PROGRAM prStation6
VAR
    SolFix : fbSingleSolRy;
    SolUpDown : fbSingleSolRy;
    SolClamp : fbSingleSolRy;
    ErrorState : BOOL;
    Autoflow : INT;
    torqueArrived1 : BOOL;
    torqueArrived2 : BOOL;
    screwL : UINT;
    oldTorqueR : LREAL;
    oldTorqueL : LREAL;
    screwR : UINT;
    TON1 : TON;
    TON2 : TON;
    ScrewLeft : fbScrewFlow;
    ScrewRight : fbScrewFlow;
    TON3 : TON;
END_VAR
VAR_EXTERNAL
    HMIPB_SOL_S5_Fix : BOOL;
    AutoStatus : bool;
    SNR_Index : BOOL;
    RY_Index : BOOL;
    SOL_S5_Fix : BOOL;
    HMIPB_SOL_S5_UpDown : BOOL;
    SOL_S5_UpDown : BOOL;
    HMIPB_SOL_S5_Clamp : BOOL;
    SOL_S5_Clamp : BOOL;
    HMIPB_SOL_S6_Fix : BOOL;
    SOL_S6_Feed : BOOL;
    SOL_S6_Fix : BOOL;
    HMIPB_SOL_S6_UpDown : BOOL;
    SOL_S6_UpDown : BOOL;
    HMIPB_SOL_S6_Clamp : BOOL;
    SOL_S6_Clamp : BOOL;
    Error_PB_Estop1 : BOOL;
    Error_PB_Estop2 : BOOL;
    Error_LS_S6_FixBack : BOOL;
    Error_LS_S6_FixOut : BOOL;
    Error_LS_S6_UpDownBack : BOOL;
    Error_LS_S6_UpDownOut : BOOL;
    IndexData6 : StationRecord;
    SystemReadyStatus : bool;
    MachineRunStatus : bool;
    HMI_ScrewTorque_St5_L : LREAL;
    HMI_ScrewSpeed_St5_L : LREAL;
    HMI_ScrewTorque_St5_R : LREAL;
    HMI_ScrewSpeed_St5_R : LREAL;
    HMIShow_CurrentTorque : ARRAY[0..3] OF LREAL;
    HMIPB_ServoStopAxisLSt5 : BOOL;
    HMIPB_ServoStopAxisRSt5 : BOOL;
    HMIPB_FW_AxisLSt5 : BOOL;
    HMIPB_FW_AxisRSt5 : BOOL;
    ScrewStartFlag : ARRAY[0..3] OF bool;
    HMI_ScrewTorque_St6_R : LREAL;
    HMI_ScrewTorque_St6_L : LREAL;
    HMI_ScrewSpeed_St6_R : LREAL;
    HMI_ScrewSpeed_St6_L : LREAL;
    HMIPB_FW_AxisLSt6 : BOOL;
    HMIPB_FW_AxisRSt6 : BOOL;
    LS_S6_UpDownOut : BOOL;
    LS_S6_UpDownBack : BOOL;
    SNR_S6_R_Check : BOOL;
    HMIPB_RW_AxisRSt6 : BOOL;
    HMIShow_CurrentSpeed : ARRAY[0..3] OF LREAL;
    LS_S6_FixBack : BOOL;
    SNR_S6_L_Check : BOOL;
    HMIPB_RW_AxisLSt6 : BOOL;
    LS_S2_MoveBack : BOOL;
    FeedStartFlag : ARRAY[0..1] OF bool;
    OBJScrewInClip : ARRAY[0..3] OF INT;
END_VAR
VAR_EXTERNAL CONSTANT
    MC_AxisLSt5 : _sAXIS_REF;
    MC_AxisLSt6 : _sAXIS_REF;
    MC_AxisRSt6 : _sAXIS_REF;
END_VAR
VAR_EXTERNAL
    ScrewStartS6LFW : BOOL;
    ScrewStartS6LRW : BOOL;
    ScrewStartS6RFW : BOOL;
    ScrewStartS6RRW : BOOL;
    HMI_BackOutTorque_St6_L : LREAL;
    HMI_BackOutTorque_St6_R : LREAL;
    Error_SNR_S6_L_Feed : BOOL;
    Error_SNR_S6_R_Feed : BOOL;
    HMI_LimitAngle_St6_L : LREAL;
    HMIShow_CurrentPosition : ARRAY[0..3] OF LREAL;
    HMI_LimitAngle_St6_R : LREAL;
    ResetAddress : ARRAY[0..3] OF bool;
    HMI_BackOutAngle_St6_L : LREAL;
    HMI_BackOutAngle_St6_R : LREAL;
    BackoutBusy : ARRAY[0..3] OF BOOL;
    BackoutStart : ARRAY[0..3] OF BOOL;
    HMI_NoScrewAngle_St6_L : LREAL;
    HMI_NoScrewAngle_St6_R : LREAL;
    HMI_Find_St6_L : LINT;
    HMI_Find_St6_R : LINT;
END_VAR
SolFix(
	inPushButton:=HMIPB_SOL_S6_Fix,
	inAutoStatus:=AutoStatus,
	inAutoFlowSet:=Autoflow=2,
	inAutoFlowReset:=Autoflow=4 OR ErrorState,
	inInterLockBack:=TRUE,
	inInterLockOut:=SNR_Index AND NOT(RY_Index),
	outSol=>SOL_S6_Fix);
SolUpDown(
	inPushButton:=HMIPB_SOL_S6_UpDown,
	inAutoStatus:=AutoStatus,
	inAutoFlowSet:=Autoflow=2,
	inAutoFlowReset:=Autoflow=4 OR ErrorState,
	inInterLockBack:=TRUE,
	inInterLockOut:=SNR_Index AND NOT(RY_Index),
	outSol=>SOL_S6_UpDown);
SolClamp(
	inPushButton:=HMIPB_SOL_S6_Clamp,
	inAutoStatus:=AutoStatus,
	inAutoFlowSet:=SOL_S6_UpDown AND LS_S6_UpDownOut AND AutoStatus AND (screwR>=2 AND screwR<20 AND screwL>=2 AND screwL<20),
	inAutoFlowReset:=(LS_S6_UpDownBack AND NOT(SOL_S6_UpDown) AND AutoStatus) OR ErrorState,
	inInterLockBack:=TRUE,
	inInterLockOut:=TRUE,
	outSol=>SOL_S6_Clamp);
TON3(In:=SOL_S6_UpDown AND LS_S6_UpDownOut AND AutoStatus,PT:=t#500ms);
(*************************************************************************************************************)
(*EStOP and Error*)
IF (Error_PB_Estop1 OR Error_PB_Estop2) AND NOT(IndexData6.OKFlag_3[6]) THEN
	IndexData6.NGFlag_3[6]:=TRUE;
	IndexData6.ErrorRecordData[6]:=1;
END_IF;
IF (Error_PB_Estop1 OR Error_PB_Estop2) AND NOT(IndexData6.OKFlag_1[6]) THEN
	IndexData6.NGFlag_1[6]:=TRUE;
	IndexData6.ErrorRecordData[6]:=1;
END_IF;
IF ErrorState AND NOT(IndexData6.OKFlag_3[6]) THEN
	IndexData6.NGFlag_3[6]:=TRUE;
	IndexData6.ErrorRecordData[6]:=2;
END_IF;
IF ErrorState AND NOT(IndexData6.OKFlag_1[6]) THEN
	IndexData6.NGFlag_1[6]:=TRUE;
	IndexData6.ErrorRecordData[6]:=2;
END_IF;
(*本站狀態判斷*)
IF (IndexData6.OKFlag_3[6] OR IndexData6.NGFlag_3[6]) AND
	(IndexData6.OKFlag_1[6] OR IndexData6.NGFlag_1[6])
	THEN
	IndexData6.FinishFlag[6]:=TRUE;
END_IF;
(*前站判斷*)
IF IndexData6.NGFlag_3[3] OR NOT(IndexData6.OKFlag_3[3]) THEN
	IndexData6.NGFlag_3[6]:=TRUE;
END_IF;
IF IndexData6.NGFlag_1[3] OR NOT(IndexData6.OKFlag_1[3]) THEN
	IndexData6.NGFlag_1[6]:=TRUE;
END_IF;
(*異常*)
ErrorState:=
Error_LS_S6_FixBack OR
Error_LS_S6_FixOut OR
Error_LS_S6_UpDownBack OR
Error_LS_S6_UpDownOut;
//*********************************自動********************************************
//****************************power on=0
IF NOT(SystemReadyStatus) OR ErrorState OR Error_PB_Estop1 OR Error_PB_Estop2 OR NOT(AutoStatus) THEN
	Autoflow:=0;
END_IF;
//****************************idle=1
IF AutoFlow=0 AND NOT(NOT(SystemReadyStatus) OR ErrorState OR Error_PB_Estop1 OR Error_PB_Estop2 OR NOT(AutoStatus)) THEN
	AutoFlow:=1;
END_IF;
IF Autoflow=4 AND screwL=1 AND screwR=1 AND LS_S6_FixBack AND LS_S6_UpDownBack THEN
	SOL_S6_Clamp:=FALSE;
	Autoflow:=1;
END_IF;
//****************************定位出,向下,鎖付開始=2
IF AutoFlow=1 AND
	NOT(FeedStartFlag[1]) AND
	NOT(Error_SNR_S6_L_Feed) AND
	NOT(Error_SNR_S6_R_Feed) AND
	NOT(SOL_S6_Feed) AND
	SNR_Index AND
	NOT(RY_Index) AND
	MachineRunStatus AND
	NOT(IndexData6.FinishFlag[6]) THEN
	ScrewStartFlag[2]:=TRUE;
	ScrewStartFlag[3]:=TRUE;
	Autoflow:=2;
END_IF;
//****************************鎖付OK=3
IF Autoflow=2 AND screwL=8 THEN//鎖付OK
	ScrewStartFlag[2]:=FALSE;
	IndexData6.OKFlag_3[6]:=TRUE;
END_IF;
IF Autoflow=2 AND screwL=9999 THEN//鎖付NG
	ScrewStartFlag[2]:=FALSE;
	IndexData6.NGFlag_3[6]:=TRUE;
END_IF;
IF Autoflow=2 AND screwR=8 THEN//鎖付OK
	ScrewStartFlag[3]:=FALSE;
	IndexData6.OKFlag_1[6]:=TRUE;
END_IF;
IF Autoflow=2 AND screwR=9999 THEN//鎖付NG
	ScrewStartFlag[3]:=FALSE;
	IndexData6.NGFlag_1[6]:=TRUE;
END_IF;
IF Autoflow=2 AND IndexData6.FinishFlag[6] THEN
	Autoflow:=3;
END_IF;
//****************************向上,定位回=4
IF Autoflow=3 AND LS_S6_UpDownOut AND NOT(ScrewStartFlag[2]) AND NOT(ScrewStartFlag[3]) THEN
	Autoflow:=4;
END_IF;
IF LS_S6_UpDownOut AND SOL_S6_UpDown AND AutoStatus THEN
	FeedStartFlag[1]:=TRUE;
END_IF;
ScrewLeft(
	inStartFlag:=ScrewStartFlag[2],
	inCheckSensor:=SNR_S6_L_Check,
	inStopFlag:= MC_AxisLSt6.Status.Standstill,
	inBackoutBusy:=BackoutBusy[2],
	inCMDTorque:=HMI_BackOutTorque_St6_L,
	inCMDAddress:=HMI_LimitAngle_St6_L,
	inNoScrewSetAngle:=HMI_NoScrewAngle_St6_L,
	inFindTime:=HMI_Find_St6_L,
	inTorqueValue:=HMIShow_CurrentTorque[2],
	inAddressValue:=HMIShow_CurrentPosition[2],
	outFW=>ScrewStartS6LFW,
	outRW=>ScrewStartS6LRW,
	outBackout=>BackoutStart[2],
	outFlowNo=> screwL,
	outResetAddress=>ResetAddress[2],
	inoutTorque:= HMI_ScrewTorque_St6_L);
ScrewRight(
	inStartFlag:=ScrewStartFlag[3],
	inCheckSensor:=SNR_S6_R_Check,
	inStopFlag:= MC_AxisRSt6.Status.Standstill,
	inBackoutBusy:=BackoutBusy[3],
	inCMDTorque:=HMI_BackOutTorque_St6_R,
	inCMDAddress:=HMI_LimitAngle_St6_R,
	inNoScrewSetAngle:=HMI_NoScrewAngle_St6_R,
	inFindTime:=HMI_Find_St6_R,
	inTorqueValue:=HMIShow_CurrentTorque[3],
	inAddressValue:=HMIShow_CurrentPosition[3],
	outFW=>ScrewStartS6RFW,
	outRW=>ScrewStartS6RRW,
	outBackout=>BackoutStart[3],
	outFlowNo=> screwR,
	outResetAddress=>ResetAddress[3],
	inoutTorque:= HMI_ScrewTorque_St6_R);
END_PROGRAM

FUNCTION fIndexDataChange : BOOL
VAR_EXTERNAL
    IndexData8 : StationRecord;
    IndexData7 : StationRecord;
    IndexData6 : StationRecord;
    IndexData5 : StationRecord;
    IndexData4 : StationRecord;
    IndexData3 : StationRecord;
    IndexData2 : StationRecord;
    IndexData1 : StationRecord;
    IndexData0 : StationRecord;
END_VAR
IndexData8:=IndexData7;
IndexData7:=IndexData6;
IndexData6:=IndexData5;
IndexData5:=IndexData4;
IndexData4:=IndexData3;
IndexData3:=IndexData2;
IndexData2:=IndexData1;
IndexData1:=IndexData0;
END_FUNCTION

FUNCTION_BLOCK fbBowlFeeder
VAR
    AutoFlow : INT;
    TON_Auto1 : TON;
    TON_Auto2 : TON;
    TON_Auto3 : TON;
    tItemNotExistDelayTime : TIME;
    tItemExistTime : TIME;
    tItemNotExistErrorTime : TIME;
END_VAR
VAR_INPUT
    bFullSNR : BOOL;
    iItemNotExistDelayTime : LINT;
    iItemExistTime : LINT;
    iItemNotExistErrorTime : LINT;
END_VAR
VAR_OUTPUT
    bFullRY : BOOL;
    bFullSNRError : BOOL;
END_VAR
VAR_EXTERNAL
    SystemReadyStatus : BOOL;
END_VAR
(******************************************************************
程式:振動筒程序
作者:蔡相偉
版本資訊:v1.0		2016/4/16
******************************************************************)
//時間轉換
tItemNotExistDelayTime:=NanoSecToTime(In:=iItemNotExistDelayTime*100000000);
tItemExistTime:=NanoSecToTime(In:=iItemExistTime*100000000);
tItemNotExistErrorTime:=NanoSecToTime(In:=iItemNotExistErrorTime*100000000);
(*流程*)
(*PowerOn=0*)
IF NOT(SystemReadyStatus) THEN
	AutoFlow:=0;
END_IF;

(*Idle=1*)
IF AutoFlow=0 AND SystemReadyStatus THEN
	AutoFlow:=1;
END_IF;

IF AutoFlow=3 THEN
	AutoFlow:=1;
END_IF;

(*振動筒起振=2*)
TON_Auto1(IN:=AutoFlow=1 AND NOT(bFullSNR) , PT:=tItemNotExistDelayTime);
IF AutoFlow=1 AND TON_Auto1.Q THEN
	AutoFlow:=2;
END_IF;

(*振動筒停振=3*)
TON_Auto2(IN:=AutoFlow=2 AND bFullSNR , PT:=tItemExistTime);
TON_Auto3(IN:=NOT(bFullSNR) AND bFullRY, PT:=tItemNotExistErrorTime);
IF AutoFlow=2 AND TON_Auto2.Q THEN
	AutoFlow:=3;
END_IF;
(******************************************************************)
(*輸出*)
(*振動筒繼電器*)
IF AutoFlow=2 THEN
	bFullRY:=TRUE;
	ELSE
	bFullRY:=FALSE;
END_IF;
(*振動筒滿料異常*)
IF AutoFlow=2 AND (TON_Auto3.Q) THEN
	bFullSNRError:=TRUE;
	ELSE
	bFullSNRError:=FALSE;
END_IF;
END_FUNCTION_BLOCK

FUNCTION_BLOCK fbSingleSolRy
VAR
    solStatus : BOOL;
    R_TRIG1 : R_TRIG;
END_VAR
VAR_INPUT
    inPushButton : BOOL;
    inAutoStatus : BOOL;
    inAutoFlowSet : BOOL;
    inAutoFlowReset : BOOL;
    inInterLockBack : BOOL;
    inInterLockOut : BOOL;
END_VAR
VAR_OUTPUT
    outSol : BOOL;
END_VAR
(*電磁閥*)
R_TRIG1(Clk:=inPushButton AND NOT(inAutoStatus));
(*SET*)
IF ((R_TRIG1.Q AND NOT(solStatus)) OR inAutoFlowSet) AND inInterLockOut THEN
	outSol:=TRUE;
END_IF;
(*RESET*)
IF ((R_TRIG1.Q AND (solStatus)) OR inAutoFlowReset) AND inInterLockBack THEN
	outSol:=FALSE;
END_IF;
(*STATUS*)
solStatus:=outSol;
END_FUNCTION_BLOCK

FUNCTION_BLOCK fbErrorSOL_S
VAR
    TON_1 : TON;
    TON_2 : TON;
END_VAR
VAR_INPUT
    bAutoStatus : BOOL;
    bResetPB : BOOL;
    bSOL : BOOL;
    bBackLS : BOOL;
    bOutLS : BOOL;
END_VAR
VAR_OUTPUT
    bErrorStatus_Back : BOOL;
    bErrorStatus_Out : BOOL;
END_VAR
IF bAutoStatus AND NOT(bResetPB) THEN
	(*歸磁簧開關*)
	TON_1(IN:=(NOT(bSOL) AND NOT(bBackLS)) OR ((bSOL) AND bBackLS), PT:=t#2s);
	IF TON_1.Q THEN
		bErrorStatus_Back:=TRUE;
	END_IF;
	(*出磁簧開關*)
	TON_2(IN:=(NOT(bSOL) AND (bOutLS)) OR ((bSOL) AND NOT(bOutLS)), PT:=t#2s);
	IF TON_2.Q THEN
		bErrorStatus_Out:=TRUE;
	END_IF;
END_IF;
IF bResetPB THEN
	bErrorStatus_Back:=FALSE;
	bErrorStatus_Out:=FALSE;
END_IF;
END_FUNCTION_BLOCK

FUNCTION_BLOCK fbErrorSOL_D
VAR
    TON_1 : TON;
    TON_2 : TON;
END_VAR
VAR_INPUT
    bAutoStatus : BOOL;
    bResetPB : BOOL;
    bBackSOL : BOOL;
    bOutSOL : BOOL;
    bBackLS : BOOL;
    bOutLS : BOOL;
END_VAR
VAR_OUTPUT
    bErrorStatus_Back : BOOL;
    bErrorStatus_Out : BOOL;
END_VAR
IF bAutoStatus AND NOT(bResetPB) THEN
	(*歸磁簧開關*)
	TON_1(IN:=bBackSOL AND NOT(bBackLS), PT:=t#4s);
	IF TON_1.Q THEN
		bErrorStatus_Back:=TRUE;
	END_IF;
	(*出磁簧開關*)
	TON_2(IN:=bOutSOL AND NOT(bOutLS), PT:=t#4s);
	IF TON_2.Q THEN
		bErrorStatus_Out:=TRUE;
	END_IF;
END_IF;
IF bResetPB THEN
	bErrorStatus_Back:=FALSE;
	bErrorStatus_Out:=FALSE;
END_IF;
END_FUNCTION_BLOCK

FUNCTION_BLOCK fbCheckScrew_Clamp
VAR
    R_TRIG1 : R_TRIG;
    R_TRIG2 : R_TRIG;
    F_TRIG1 : F_TRIG;
END_VAR
VAR_INPUT
    inClearSingle : BOOL;
    inFeedSNR : BOOL;
    inBlowSOL : BOOL;
    inReset : BOOL;
END_VAR
VAR_OUTPUT
    outError : BOOL;
END_VAR
VAR_IN_OUT
    inoutScrewInClip : INT;
END_VAR
R_TRIG1(CLK:= inClearSingle);
R_TRIG2(CLK:= inFeedSNR);
F_TRIG1(Clk:=inBlowSOL);

IF R_TRIG2.Q THEN
	inoutScrewInClip:=inoutScrewInClip+1;
END_IF;

IF R_TRIG1.Q THEN
	inoutScrewInClip:=0;
END_IF;

IF F_TRIG1.Q AND inoutScrewInClip<=0 THEN
	outError:=TRUE;
END_IF;
IF inReset THEN
	outError:=FALSE;
END_IF;
END_FUNCTION_BLOCK

FUNCTION_BLOCK fbDoubleSolRy
VAR_INPUT
    inPushBackButton : BOOL;
    inPushOutButton : BOOL;
    inAutoStatus : BOOL;
    inAutoFlowSet : BOOL;
    inAutoFlowReset : BOOL;
    inInterLockBack : BOOL;
    inInterLockOut : BOOL;
    inBackSensor : BOOL;
    inOutSensor : BOOL;
END_VAR
VAR_OUTPUT
    outBackSol : BOOL;
    outOutSol : BOOL;
END_VAR
(*Out電磁閥*)
IF (inPushOutButton OR inAutoFlowSet) AND inInterLockOut THEN
	outOutSol:=TRUE;
	outBackSol:=FALSE;
END_IF;
IF inOutSensor THEN
	outOutSol:=FALSE;
END_IF;
(*Back電磁閥*)
IF (inPushBackButton OR inAutoFlowReset) AND inInterLockBack THEN
	outOutSol:=FALSE;
	outBackSol:=TRUE;
END_IF;
IF inBackSensor THEN
	outBackSol:=FALSE;
END_IF;
END_FUNCTION_BLOCK

FUNCTION_BLOCK fbCheckScrew_Tube
VAR
    R_TRIG1 : R_TRIG;
    R_TRIG2 : R_TRIG;
    R_TRIG3 : R_TRIG;
    F_TRIG1 : F_TRIG;
END_VAR
VAR_INPUT
    inClearSingle : BOOL;
    inFeedSNR : BOOL;
    inBlowSOL : BOOL;
    inReset : BOOL;
END_VAR
VAR_OUTPUT
    outError : BOOL;
END_VAR
VAR_IN_OUT
    inoutScrewInClip : INT;
    inoutScrewInTube : INT;
END_VAR
R_TRIG1(CLK:= inClearSingle);
R_TRIG2(CLK:= inFeedSNR);
R_TRIG3(CLK:= inBlowSOL);
F_TRIG1(Clk:=inBlowSOL);

IF R_TRIG2.Q THEN
	inoutScrewInTube:=inoutScrewInTube+1;
END_IF;

(*
IF R_TRIG1.Q THEN
	inoutScrewInClip:=0;
END_IF;
*)
IF R_TRIG3.Q THEN
	inoutScrewInClip:=inoutScrewInTube;
	inoutScrewInTube:=0;
END_IF;

IF (*F_TRIG1.Q AND*) inoutScrewInClip =0 THEN
	outError:=TRUE;
ELSE
	outError:=FALSE;
END_IF;
IF inReset THEN
	inoutScrewInClip:=1;
	//outError:=FALSE;
END_IF;
END_FUNCTION_BLOCK

FUNCTION_BLOCK fbScrewFlow
VAR
    AutoFlow : INT;
    TONNG : TON;
    TON7 : TON;
    TON20 : TON;
    TON30 : TON;
    oldTorque : LREAL;
    torquecount : INT;
    sensorONFlag : BOOL;
END_VAR
VAR_INPUT
    inStartFlag : BOOL;  (* 起動 *)
    inCheckSensor : BOOL;  (* 檢查近接開關 *)
    inStopFlag : BOOL;  (* standstill *)
    inBackoutBusy : BOOL;  (* busy *)
    inCMDTorque : LREAL;  (* 退扭力 *)
    inCMDAddress : LREAL;  (* 下鎖限制角度 *)
    inNoScrewSetAngle : LREAL;  (* 無螺絲檢查角度 *)
    inFindTime : LINT;  (* 反轉時間 *)
    inTorqueValue : LREAL;  (* 扭力顯示 *)
    inAddressValue : LREAL;  (* 角度顯示 *)
END_VAR
VAR_OUTPUT
    outFW : BOOL;  (* 正轉PB *)
    outRW : BOOL;  (* 反轉PB *)
    outBackout : BOOL;  (* Backout Start *)
    outFlowNo : INT;  (* 當前流程碼 *)
    outResetAddress : BOOL;  (* HOME PB *)
END_VAR
VAR_IN_OUT
    inoutTorque : LREAL;  (* 下鎖扭力設定值 *)
END_VAR
VAR_EXTERNAL
    SystemReadyStatus : bool;
END_VAR
VAR_EXTERNAL CONSTANT
    MC_AxisLSt5 : _sAXIS_REF;
END_VAR
//power on
IF NOT(SystemReadyStatus) THEN
	AutoFlow:=0;
END_IF;
//idle
IF AutoFlow=0 AND SystemReadyStatus THEN
	AutoFlow:=1;
END_IF;
IF AutoFlow=8 AND NOT(outRW) AND NOT(inStartFlag) AND oldTorque=inoutTorque THEN
	AutoFlow:=1;
END_IF;
IF AutoFlow=9999 AND NOT(outFW) AND NOT(inStartFlag) AND oldTorque=inoutTorque  THEN
	AutoFlow:=1;
END_IF;
//反轉=30
IF AutoFlow=1 AND inStartFlag THEN
	torquecount:=0;
	oldTorque:=inoutTorque;
	outResetAddress:=TRUE;
	sensorONFlag:=FALSE;
	outRW:=TRUE;
	AutoFlow:=30;
END_IF;
//停止=31
TON30(In:=AutoFlow=30 AND outRW, PT:=NanoSecToTime(In:=inFindTime*100000000));
IF AutoFlow=30 AND TON30.Q THEN
    outRW:=FALSE;
	AutoFlow:=31;
END_IF;
//set 0 on=20
IF AutoFlow=31 AND NOT(outRW) AND inStopFlag THEN
	AutoFlow:=20;
END_IF;
//set0 off=21
TON20(In:=AutoFlow=20 AND outResetAddress,PT:=t#300ms);
IF AutoFlow=20 AND TON20.Q THEN
	outResetAddress:=FALSE;
	AutoFlow:=21;
END_IF;
//起動=2
IF AutoFlow=21 AND NOT(outResetAddress) THEN
	outFW:=TRUE;
	AutoFlow:=2;
END_IF;
//snesor到達=3
IF AutoFlow=2 AND inCheckSensor AND NOT(TONNG.Q) THEN
	AutoFlow:=3;
END_IF;
//snesor未到達=9999
TONNG(In:=AutoFlow>=2 AND AutoFlow<9000,PT:=t#6s);
IF AutoFlow>=2 AND TONNG.Q THEN
	outFW:=FALSE;
	outRW:=FALSE;
	inoutTorque:=oldTorque;
	AutoFlow:=9999;
END_IF;
IF AutoFlow=2 AND (inAddressValue>=inCMDAddress) AND oldTorque=inoutTorque THEN
	outFW:=FALSE;
	outRW:=FALSE;
	inoutTorque:=oldTorque;
	AutoFlow:=9999;
END_IF;
IF inCheckSensor THEN
	sensorONFlag:=TRUE;
END_IF;

//停止=4
IF AutoFlow=3 AND inCheckSensor THEN
	outFW:=FALSE;
	AutoFlow:=4;
END_IF;
//設定=5
IF AutoFlow=4 AND NOT(outFW) THEN
	AutoFlow:=5;
END_IF;
//反轉=6
IF AutoFlow=5 AND inStopFlag THEN
	outBackout:=TRUE;
	AutoFlow:=6;
END_IF;
//反轉中=7
IF AutoFlow=6 AND inBackoutBusy THEN
	outBackout:=FALSE;
	AutoFlow:=7;
END_IF;
//停止=8
IF AutoFlow=7 AND NOT(inBackoutBusy) AND NOT(outRW) THEN
	AutoFlow:=8;
END_IF;
outFlowNo:=AutoFlow;
END_FUNCTION_BLOCK